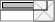
VISUALIZATION SYM_CACHE  // 55x22
VAR_IN_OUT
	m_Input_CACHE : BLOCK_ACTUATOR;
END_VAR
    Rectangle (2,2 43x6), colour toggle: (m_Input_CACHE.STATE_OFF) <> 0, invisible if: (m_Input_CACHE.STATE_ON) <> 0
    Rectangle (0,0 47x10), invisible if: NOT m_Input_CACHE.AUTOR_On_IHM OR NOT PRG_USER.ACTU_USER.MAINTENANCE, input disabled if: NOT m_Input_CACHE.AUTOR_On_IHM OR NOT PRG_User.ACTU_USER.MAINTENANCE
        tap m_Input_CACHE.M_ON
    Image (33,0 22x22), invisible if: NOT m_Input_CACHE.STATE_NOK, image: MesImages.warning
    Rectangle (0,0 47x10), invisible if: NOT m_Input_CACHE.AUTOR_Off_IHM OR NOT PRG_USER.ACTU_USER.MAINTENANCE, input disabled if: NOT m_Input_CACHE.AUTOR_Off_IHM OR NOT PRG_User.ACTU_USER.MAINTENANCE
        tap m_Input_CACHE.M_Off
END_VISUALIZATION

(* stored: Version 1.1.0.1, ProductVersion 3.1.4024.11
   Visu SYM_CACHE: Id {73b09ec1-98e0-441f-92bc-b5b41451add6} *)
